{attribute clr[Container(Layout.Stack)]}
{attribute clr[Group(Layout.GroupBox)]}
{attribute addProperty PreviousPort "Unknown"}
TYPE EtcSlaveTerminalBase_947E5A46 EXTENDS EtcSlaveBase_82538BE2 :
STRUCT
END_STRUCT
END_TYPE

(* stored: Version 1.2.0.0
   DUT EtcSlaveTerminalBase_947E5A46: Id {52cfa0ba-5632-49b0-ac0c-57ddc7e9ca2a} *)
